FUNCTION_BLOCK ABSTRACT PiperModule IMPLEMENTS IPiperModule, ISequence, IStepManager
VAR
    _piperModule : PiperModuleInternal;
    i_sequence : SequenceType;
    _sequence : Sequencer(THIS^);
    command : PLCopenCall;
END_VAR

// Copyright (c) 2024 Loupe (https://loupe.team), provided under the MIT License.

METHOD _RequestStep : BOOL
VAR_INPUT
    nextStep : ENUM;
END_VAR
// Copyright (c) 2024 Loupe (https://loupe.team), provided under the MIT License.

_piperModule.requestSubstate := nextStep;
_piperModule.response := RESPONSE_STATE.BUSY;
_piperModule.requestNumber := _piperModule.requestNumber + 1;
END_METHOD

METHOD _Reset : BOOL
// Copyright (c) 2024 Loupe (https://loupe.team), provided under the MIT License.
END_METHOD

METHOD _SequenceComplete : BOOL
// Copyright (c) 2024 Loupe (https://loupe.team), provided under the MIT License.

_piperModule.requestSubstate := 0;
_piperModule.response := RESPONSE_STATE.DONE;
END_METHOD

METHOD _SequenceError : BOOL
// Copyright (c) 2024 Loupe (https://loupe.team), provided under the MIT License.

_piperModule.requestSubstate := 0;
_piperModule.response := RESPONSE_STATE.ERROR;
END_METHOD

METHOD Aborted : BOOL
// Copyright (c) 2024 Loupe (https://loupe.team), provided under the MIT License.

i_sequence.activeTasks.Aborted();
END_METHOD

METHOD Aborting : MACHINE_STATE
// Copyright (c) 2024 Loupe (https://loupe.team), provided under the MIT License.

_piperModule.skipsSync.aborting := TRUE;
END_METHOD

METHOD AbortingAsync : MACHINE_STATE
// Copyright (c) 2024 Loupe (https://loupe.team), provided under the MIT License.

_piperModule.skipsAsync.aborting := TRUE;
END_METHOD

METHOD Booting : MACHINE_STATE
// Copyright (c) 2024 Loupe (https://loupe.team), provided under the MIT License.

_piperModule.skipsSync.booting := TRUE;
END_METHOD

METHOD BootingAsync : MACHINE_STATE
// Copyright (c) 2024 Loupe (https://loupe.team), provided under the MIT License.

_piperModule.skipsAsync.booting := TRUE;
END_METHOD

METHOD CallState : BOOL
VAR_INPUT

END_VAR
// Copyright (c) 2024 Loupe (https://loupe.team), provided under the MIT License.

THIS^.WillCall();

IF THIS^._piperModule.previousSubstate <> THIS^.CurrentSubstate THEN
    THIS^.WillChangeSubstate();
END_IF

THIS^._piperModule.previousSubstate := THIS^.CurrentSubstate;

IF Response <> RESPONSE_STATE.DONE AND RequestedSubstate <= CurrentSubstate THEN
    CASE CurrentState OF
        MACHINE_STATE.ABORTING:
            IF NOT _piperModule.skipsSync.aborting THEN
                THIS^.Aborting();
            END_IF

        MACHINE_STATE.BOOTING:
            IF NOT _piperModule.skipsSync.booting THEN
                THIS^.Booting();
            END_IF

        MACHINE_STATE.CLEARING:
            IF NOT _piperModule.skipsSync.clearing THEN
                THIS^.Clearing();
            END_IF

        MACHINE_STATE.COMPLETING:
            IF NOT _piperModule.skipsSync.completing THEN
                THIS^.COMPLETING();
            END_IF

        MACHINE_STATE.EXECUTING:
            IF NOT _piperModule.skipsSync.executing THEN
                THIS^.Executing();
            END_IF

        MACHINE_STATE.HOLDING:
            IF NOT _piperModule.skipsSync.holding THEN
                THIS^.Holding();
            END_IF

        MACHINE_STATE.RESETTING:
            IF NOT _piperModule.skipsSync.resetting THEN
                THIS^.Resetting();
            END_IF

        MACHINE_STATE.STARTING:
            IF NOT _piperModule.skipsSync.starting THEN
                THIS^.Starting();
            END_IF

        MACHINE_STATE.STOPPING:
            IF NOT _piperModule.skipsSync.stopping THEN
                THIS^.Stopping();
            END_IF

        MACHINE_STATE.SUSPENDING:
            IF NOT _piperModule.skipsSync.suspending THEN
                THIS^.Suspending();
            END_IF

        MACHINE_STATE.UNHOLDING:
            IF NOT _piperModule.skipsSync.unholding THEN
                THIS^.Unholding();
            END_IF

        MACHINE_STATE.UNSUSPENDING:
            IF NOT _piperModule.skipsSync.unsuspending THEN
                THIS^.Unsuspending();
            END_IF

    END_CASE
END_IF

THIS^.DidCall();
END_METHOD

METHOD CallStateAsync : BOOL
VAR_INPUT

END_VAR
// Copyright (c) 2024 Loupe (https://loupe.team), provided under the MIT License.

THIS^.WillCallAsync();

IF THIS^._piperModule.previousSubstateAsync <> THIS^.CurrentSubstate THEN
    THIS^.WillChangeSubstateAsync();
END_IF

THIS^._piperModule.previousSubstateAsync := THIS^.CurrentSubstate;

IF Response <> RESPONSE_STATE.DONE AND RequestedSubstate <= CurrentSubstate THEN
    CASE CurrentState OF
        MACHINE_STATE.ABORTING:
            IF NOT _piperModule.skipsAsync.aborting THEN
                THIS^.AbortingAsync();
            ELSIF _piperModule.skipsSync.aborting THEN
                _piperModule.response := RESPONSE_STATE.DONE;
            END_IF

        MACHINE_STATE.BOOTING:
            IF NOT _piperModule.skipsAsync.booting THEN
                THIS^.BootingAsync();
            ELSIF _piperModule.skipsSync.booting THEN
                _piperModule.response := RESPONSE_STATE.DONE;
            END_IF

        MACHINE_STATE.CLEARING:
            IF NOT _piperModule.skipsAsync.clearing THEN
                THIS^.ClearingAsync();
            ELSIF _piperModule.skipsSync.clearing THEN
                _piperModule.response := RESPONSE_STATE.DONE;
            END_IF

        MACHINE_STATE.COMPLETING:
            IF NOT _piperModule.skipsAsync.completing THEN
                THIS^.CompletingAsync();
            ELSIF _piperModule.skipsSync.completing THEN
                _piperModule.response := RESPONSE_STATE.DONE;
            END_IF

        MACHINE_STATE.EXECUTING:
            IF NOT _piperModule.skipsAsync.executing THEN
                THIS^.ExecutingAsync();
            ELSIF _piperModule.skipsSync.executing THEN
                _piperModule.response := RESPONSE_STATE.DONE;
            END_IF

        MACHINE_STATE.HOLDING:
            IF NOT _piperModule.skipsAsync.holding THEN
                THIS^.HoldingAsync();
            ELSIF _piperModule.skipsSync.holding THEN
                _piperModule.response := RESPONSE_STATE.DONE;
            END_IF

        MACHINE_STATE.RESETTING:
            IF NOT _piperModule.skipsAsync.resetting THEN
                THIS^.ResettingAsync();
            ELSIF _piperModule.skipsSync.resetting THEN
                _piperModule.response := RESPONSE_STATE.DONE;
            END_IF

        MACHINE_STATE.STARTING:
            IF NOT _piperModule.skipsAsync.starting THEN
                THIS^.StartingAsync();
            ELSIF _piperModule.skipsSync.starting THEN
                _piperModule.response := RESPONSE_STATE.DONE;
            END_IF

        MACHINE_STATE.STOPPING:
            IF NOT _piperModule.skipsAsync.stopping THEN
                THIS^.StoppingAsync();
            ELSIF _piperModule.skipsSync.stopping THEN
                _piperModule.response := RESPONSE_STATE.DONE;
            END_IF

        MACHINE_STATE.SUSPENDING:
            IF NOT _piperModule.skipsAsync.suspending THEN
                THIS^.SuspendingAsync();
            ELSIF _piperModule.skipsSync.suspending THEN
                _piperModule.response := RESPONSE_STATE.DONE;
            END_IF

        MACHINE_STATE.UNHOLDING:
            IF NOT _piperModule.skipsAsync.unholding THEN
                THIS^.UnholdingAsync();
            ELSIF _piperModule.skipsSync.unholding THEN
                _piperModule.response := RESPONSE_STATE.DONE;
            END_IF

        MACHINE_STATE.UNSUSPENDING:
            IF NOT _piperModule.skipsAsync.unsuspending THEN
                THIS^.UnsuspendingAsync();
            ELSIF _piperModule.skipsSync.unsuspending THEN
                _piperModule.response := RESPONSE_STATE.DONE;
            END_IF

    END_CASE
END_IF

THIS^.DidCallAsync();
END_METHOD

METHOD PRIVATE CheckStatus : BOOL
VAR
    _commandIndex : INT;
    _anyAbort : BOOL;
    _anyBusy : BOOL;
    _anyError : BOOL;
END_VAR
// Copyright (c) 2024 Loupe (https://loupe.team), provided under the MIT License.

IF NOT i_sequence.statusChecked THEN
    //We cache the is abort so that we have a consistent 
    //	status for the whole state
    i_sequence.isError := i_sequence.activeTasks.isError;
    i_sequence.isAbort := i_sequence.activeTasks.isAbort;
    i_sequence.isDone := i_sequence.activeTasks.isDone;
END_IF
END_METHOD

METHOD Clearing : MACHINE_STATE
// Copyright (c) 2024 Loupe (https://loupe.team), provided under the MIT License.

_piperModule.skipsSync.clearing := TRUE;
END_METHOD

METHOD ClearingAsync : MACHINE_STATE
// Copyright (c) 2024 Loupe (https://loupe.team), provided under the MIT License.

_piperModule.skipsAsync.clearing := TRUE;
END_METHOD

METHOD Completing : MACHINE_STATE
// Copyright (c) 2024 Loupe (https://loupe.team), provided under the MIT License.

_piperModule.skipsSync.completing := TRUE;
END_METHOD

METHOD CompletingAsync : MACHINE_STATE
// Copyright (c) 2024 Loupe (https://loupe.team), provided under the MIT License.

_piperModule.skipsAsync.completing := TRUE;
END_METHOD

PROPERTY CurrentState : MACHINE_STATE
GET
// Copyright (c) 2024 Loupe (https://loupe.team), provided under the MIT License.

CurrentState := _piperModule.machine.PackMLState;
END_GET
END_PROPERTY

PROPERTY CurrentStep : ENUM
GET
// Copyright (c) 2024 Loupe (https://loupe.team), provided under the MIT License.

CurrentStep := ULINT_TO_UDINT(_piperModule.machine.Substate);
END_GET
END_PROPERTY

PROPERTY CurrentSubstate : ULINT
GET
// Copyright (c) 2024 Loupe (https://loupe.team), provided under the MIT License.

CurrentSubstate := _piperModule.machine.Substate;
END_GET
END_PROPERTY

METHOD DidCall : BOOL
VAR_INPUT
END_VAR
// Copyright (c) 2024 Loupe (https://loupe.team), provided under the MIT License.
END_METHOD

METHOD DidCallAsync : BOOL
VAR_INPUT
END_VAR
// Copyright (c) 2024 Loupe (https://loupe.team), provided under the MIT License.
END_METHOD

METHOD DoStep : ENUM
VAR
END_VAR
// Copyright (c) 2024 Loupe (https://loupe.team), provided under the MIT License.

DoStep := _sequence.DoStep();
END_METHOD

METHOD Errored : BOOL
VAR_INPUT
    ID : INT;
END_VAR
// Copyright (c) 2024 Loupe (https://loupe.team), provided under the MIT License.

i_sequence.activeTasks.Errored(ID);
END_METHOD

METHOD Executing : MACHINE_STATE
// Copyright (c) 2024 Loupe (https://loupe.team), provided under the MIT License.

_piperModule.skipsSync.executing := TRUE;
END_METHOD

METHOD ExecutingAsync : MACHINE_STATE
// Copyright (c) 2024 Loupe (https://loupe.team), provided under the MIT License.

_piperModule.skipsAsync.executing := TRUE;
END_METHOD

METHOD FB_init : BOOL
VAR_INPUT
    bInitRetains : BOOL; // if TRUE, the retain variables are initialized (warm start / cold start)
    bInCopyCode : BOOL; // if TRUE, the instance afterwards gets moved into the copy code (online change)
    machineIn : REFERENCE TO Piper;
    //	context : IPluginRunner;
END_VAR
// Copyright (c) 2024 Loupe (https://loupe.team), provided under the MIT License.
RegisterToMachine(machineIn);
//THIS^.setContext( context );
END_METHOD

METHOD Finished : BOOL
// Copyright (c) 2024 Loupe (https://loupe.team), provided under the MIT License.

i_sequence.activeTasks.Finished();
END_METHOD

METHOD Holding : MACHINE_STATE
// Copyright (c) 2024 Loupe (https://loupe.team), provided under the MIT License.

_piperModule.skipsSync.holding := TRUE;
END_METHOD

METHOD HoldingAsync : MACHINE_STATE
// Copyright (c) 2024 Loupe (https://loupe.team), provided under the MIT License.

_piperModule.skipsAsync.holding := TRUE;
END_METHOD

PROPERTY IsAbort : BOOL
GET
// Copyright (c) 2024 Loupe (https://loupe.team), provided under the MIT License.

CheckStatus();
IsAbort := i_sequence.isAbort;
END_GET
END_PROPERTY

PROPERTY IsDone : BOOL
GET
// Copyright (c) 2024 Loupe (https://loupe.team), provided under the MIT License.

CheckStatus();
IsDone := i_sequence.isDone;
END_GET
END_PROPERTY

PROPERTY IsError : BOOL
GET
// Copyright (c) 2024 Loupe (https://loupe.team), provided under the MIT License.

CheckStatus();
IsError := i_sequence.isError;
END_GET
END_PROPERTY

METHOD OnAbort : BOOL
VAR_INPUT
    nextStep : ENUM;
END_VAR
// Copyright (c) 2024 Loupe (https://loupe.team), provided under the MIT License.

OnAbort := _sequence.OnAbort(nextStep);
END_METHOD

METHOD OnEntry : BOOL
VAR_INPUT
END_VAR
// Copyright (c) 2024 Loupe (https://loupe.team), provided under the MIT License.

OnEntry := _sequence.OnEntry();
END_METHOD

METHOD OnError : BOOL
VAR_INPUT
    nextStep : ENUM;
END_VAR
// Copyright (c) 2024 Loupe (https://loupe.team), provided under the MIT License.

OnError := _sequence.OnError(nextStep);
END_METHOD

METHOD OnExit : BOOL
VAR_INPUT
END_VAR
// Copyright (c) 2024 Loupe (https://loupe.team), provided under the MIT License.

OnExit := _sequence.OnExit();
END_METHOD

METHOD OnFailure : BOOL
VAR_INPUT
    nextStep : ENUM;
END_VAR
// Copyright (c) 2024 Loupe (https://loupe.team), provided under the MIT License.

OnFailure := _sequence.OnFailure(nextStep);
END_METHOD

METHOD OnSuccess : BOOL
VAR_INPUT
    nextStep : ENUM;
END_VAR
// Copyright (c) 2024 Loupe (https://loupe.team), provided under the MIT License.

OnSuccess := _sequence.OnSuccess(nextStep);
END_METHOD

METHOD RegisterToMachine : DINT
VAR_INPUT
    machineIn : REFERENCE TO Piper;
END_VAR
VAR
END_VAR
// Copyright (c) 2024 Loupe (https://loupe.team), provided under the MIT License.
IF NOT _piperModule.registered THEN
    _piperModule.registered := TRUE;
    _piperModule.machine REF= machineIn;
    _piperModule.machine.RegisterSubmodule(THIS^);
END_IF
END_METHOD

{warning 'add property implementation'}
PROPERTY RequestedSubstate : ULINT
GET
// Copyright (c) 2024 Loupe (https://loupe.team), provided under the MIT License.

RequestedSubstate := _piperModule.requestSubstate;
END_GET
END_PROPERTY

PROPERTY RequestNumber : DINT
GET
// Copyright (c) 2024 Loupe (https://loupe.team), provided under the MIT License.

RequestNumber := _piperModule.requestNumber;
END_GET
END_PROPERTY

METHOD RequestStep : BOOL
VAR_INPUT
    nextStep : ENUM;
END_VAR
// Copyright (c) 2024 Loupe (https://loupe.team), provided under the MIT License.

RequestStep := _sequence.requestStep(nextStep);
END_METHOD

METHOD RequestStepClear : BOOL
VAR_INPUT
    nextStep : ENUM;
END_VAR
// Copyright (c) 2024 Loupe (https://loupe.team), provided under the MIT License.

RequestStepClear := _sequence.requestStepClear(nextStep);
END_METHOD

METHOD Resetting : BOOL
// Copyright (c) 2024 Loupe (https://loupe.team), provided under the MIT License.

_piperModule.skipsSync.resetting := TRUE;
END_METHOD

METHOD ResettingAsync : BOOL
// Copyright (c) 2024 Loupe (https://loupe.team), provided under the MIT License.

_piperModule.skipsAsync.resetting := TRUE;
END_METHOD

PROPERTY Response : RESPONSE_STATE
GET
// Copyright (c) 2024 Loupe (https://loupe.team), provided under the MIT License.

Response := _piperModule.response;
END_GET
END_PROPERTY

METHOD Run : BOOL
// Copyright (c) 2024 Loupe (https://loupe.team), provided under the MIT License.

THIS^.CallState();
END_METHOD

METHOD SequenceAbort : BOOL
VAR_INPUT
    ErrorCode : DINT;
    ErrorMessage : STRING;
END_VAR
// Copyright (c) 2024 Loupe (https://loupe.team), provided under the MIT License.

SequenceAbort := _sequence.sequenceAbort(ErrorCode, ErrorMessage);
END_METHOD

METHOD SequenceComplete : BOOL
VAR_INPUT
END_VAR
// Copyright (c) 2024 Loupe (https://loupe.team), provided under the MIT License.

SequenceComplete := _sequence.sequenceComplete();
END_METHOD

METHOD SequenceError : BOOL
VAR_INPUT
    ErrorCode : DINT;
    ErrorMessage : STRING;
END_VAR
// Copyright (c) 2024 Loupe (https://loupe.team), provided under the MIT License.

SequenceError := _sequence.sequenceError(ErrorCode, ErrorMessage);
END_METHOD

METHOD SetContext : BOOL
VAR_INPUT
    context : IPluginRunner;
END_VAR
// Copyright (c) 2024 Loupe (https://loupe.team), provided under the MIT License.
_piperModule.context := context;
context.RegisterPlugin(THIS^);
END_METHOD

METHOD SetState : BOOL
VAR_INPUT
END_VAR
// Copyright (c) 2024 Loupe (https://loupe.team), provided under the MIT License.

_piperModule.requestSubstate := 0;
_piperModule.response := RESPONSE_STATE.UNDEFINED;
_sequence.startSequence();
END_METHOD

METHOD Start : BOOL
VAR_INPUT
    Command : IPLCopenCommand;
END_VAR
// Copyright (c) 2024 Loupe (https://loupe.team), provided under the MIT License.

IF i_sequence.activeTasks.Start(Command) = 0 THEN
    //TODO: All out of commands.. Throw an error
    SequenceError(10000, 'Too Many Commands in 1 step');
    Start := FALSE;
ELSE
    Start := TRUE;
END_IF
END_METHOD

METHOD Starting : MACHINE_STATE
// Copyright (c) 2024 Loupe (https://loupe.team), provided under the MIT License.

_piperModule.skipsSync.starting := TRUE;
END_METHOD

METHOD StartingAsync : MACHINE_STATE
// Copyright (c) 2024 Loupe (https://loupe.team), provided under the MIT License.

_piperModule.skipsAsync.starting := TRUE;
END_METHOD

METHOD StartSequence : BOOL
// Copyright (c) 2024 Loupe (https://loupe.team), provided under the MIT License.

RequestStep(0);
END_METHOD

METHOD StateCompletePending : BOOL
VAR_INPUT
END_VAR
// Copyright (c) 2024 Loupe (https://loupe.team), provided under the MIT License.

_piperModule.response := RESPONSE_STATE.DONE_PENDING;
END_METHOD

METHOD StateErrored : BOOL
VAR_INPUT
END_VAR
// Copyright (c) 2024 Loupe (https://loupe.team), provided under the MIT License.

_piperModule.response := RESPONSE_STATE.ERROR;
END_METHOD

METHOD Stopping : MACHINE_STATE
// Copyright (c) 2024 Loupe (https://loupe.team), provided under the MIT License.

_piperModule.skipsSync.stopping := TRUE;
END_METHOD

METHOD StoppingAsync : MACHINE_STATE
// Copyright (c) 2024 Loupe (https://loupe.team), provided under the MIT License.

_piperModule.skipsAsync.stopping := TRUE;
END_METHOD

METHOD Suspending : MACHINE_STATE
// Copyright (c) 2024 Loupe (https://loupe.team), provided under the MIT License.

_piperModule.skipsSync.suspending := TRUE;
END_METHOD

METHOD SuspendingAsync : MACHINE_STATE
// Copyright (c) 2024 Loupe (https://loupe.team), provided under the MIT License.

_piperModule.skipsAsync.suspending := TRUE;
END_METHOD

METHOD Undefined : MACHINE_STATE
// Copyright (c) 2024 Loupe (https://loupe.team), provided under the MIT License.

_piperModule.response := RESPONSE_STATE.NO_IMPL;
END_METHOD

METHOD UndefinedAsync : MACHINE_STATE
// Copyright (c) 2024 Loupe (https://loupe.team), provided under the MIT License.
END_METHOD

METHOD Unholding : MACHINE_STATE
// Copyright (c) 2024 Loupe (https://loupe.team), provided under the MIT License.

_piperModule.skipsSync.unholding := TRUE;
END_METHOD

METHOD UnholdingAsync : MACHINE_STATE
// Copyright (c) 2024 Loupe (https://loupe.team), provided under the MIT License.

_piperModule.skipsAsync.unholding := TRUE;
END_METHOD

METHOD Unsuspending : MACHINE_STATE
// Copyright (c) 2024 Loupe (https://loupe.team), provided under the MIT License.

_piperModule.skipsSync.unsuspending := TRUE;
END_METHOD

METHOD UnsuspendingAsync : MACHINE_STATE
// Copyright (c) 2024 Loupe (https://loupe.team), provided under the MIT License.

_piperModule.skipsAsync.unsuspending := TRUE;
END_METHOD

METHOD WillCall : BOOL
VAR_INPUT
END_VAR
// Copyright (c) 2024 Loupe (https://loupe.team), provided under the MIT License.
END_METHOD

METHOD WillCallAsync : BOOL
VAR_INPUT
END_VAR
// Copyright (c) 2024 Loupe (https://loupe.team), provided under the MIT License.
END_METHOD

METHOD WillChangeSubstate : BOOL
VAR_INPUT
END_VAR
// Copyright (c) 2024 Loupe (https://loupe.team), provided under the MIT License.
END_METHOD

METHOD WillChangeSubstateAsync : BOOL
VAR_INPUT
END_VAR
// Copyright (c) 2024 Loupe (https://loupe.team), provided under the MIT License.
END_METHOD

END_FUNCTION_BLOCK

(* stored: Version 1.1.0.1
   POU PiperModule: Id {a49f2d62-e1fb-48a5-85f3-63c6ca0008b5}, SpecialFunc None
   Folder Handshake: Id {4c5f2be6-50e2-4221-9823-927772de0d3d}
   Folder PackML: Id {103dd83a-b3d9-4ad0-8c08-4f9980ee4239}
   Folder PackMLAsync: Id {8d7f90b0-8dd2-435c-bd8c-5cc1b1fbb6fd}
   Folder PLCopen: Id {64089310-c2b2-409b-a0ee-99363ab988ef}
   Folder Sequence: Id {8453be56-3070-4e48-be57-e6bddaa0c622}
   Folder callbacks: Id {778d4fd5-4d6a-48ab-b39c-efcbe9f36276}
   Folder StateControl: Id {6b001fba-3153-4b1f-932c-0a719f676126}
   Folder Setup: Id {eeb68776-0e62-46f1-9ad5-da0f6ad004d6}
   Folder StepManager: Id {48dc10ce-7eca-4656-a440-fb808be36402}
   Method _RequestStep: Id {f4f6af93-0cb3-42b4-9ca9-21e1cca56843}
   Method _Reset: Id {e5c4fbde-1df8-48bc-9d3c-c9ad0b85ba57}
   Method _SequenceComplete: Id {93d7990e-83cd-41da-874b-7bcab730bc0b}
   Method _SequenceError: Id {d8c3afc4-de9e-411e-b9c4-728f5280910b}
   Method Aborted: Id {bfc1fdac-439e-4113-ad1e-f9923d22408a}
   Method Aborting: Id {f8a973b9-f9f6-410e-b5c1-d3a51e04d7ba}
   Method AbortingAsync: Id {cec06300-8aeb-4e42-9276-4c70e9317f91}
   Method Booting: Id {8c4cd35b-8b79-4b7d-b8d1-be00bdf7a998}
   Method BootingAsync: Id {9ce4a9c1-65bb-4257-8807-dd0b22b34a12}
   Method CallState: Id {8c189048-9fa3-4697-bf51-2b2792a9dbd0}
   Method CallStateAsync: Id {e1b90424-eb8a-4298-af7b-9ebf7a18fd7f}
   Method CheckStatus: Id {86f2cd85-d973-4227-9da3-ee4c3ed52cb2}
   Method Clearing: Id {7bee31c9-141c-4358-8aca-33cad167ec8c}
   Method ClearingAsync: Id {f3e36a82-f507-456f-b94b-64cf7681213f}
   Method Completing: Id {a413a61c-6ca7-4fd3-9296-7d7fa43065a1}
   Method CompletingAsync: Id {a25aad53-5324-4bcd-8931-defa299aa789}
   Property CurrentState: Id {a9acd7a7-2c0b-4c94-b2f1-fd8eff4ca549}
   Get Get: Id {f9b34f5c-82e0-4f78-84c5-ae373d09c208}
   Property CurrentStep: Id {674ced14-3f04-4cfd-8fdd-09d4136719f6}
   Get Get: Id {bf1b5077-fd19-49ed-99c4-4f1808c79d8e}
   Property CurrentSubstate: Id {88b27a69-ed23-442a-a3ec-53bdad984f5d}
   Get Get: Id {b3583fbe-c993-43b1-b2df-a70ec57198b2}
   Method DidCall: Id {5d73cdfc-bb8e-4ce5-9441-fb7bff95dddb}
   Method DidCallAsync: Id {1c612e8f-0b57-4feb-b3a0-8272535d9fbf}
   Method DoStep: Id {2460656a-9a34-4d02-b4bf-86513714621e}
   Method Errored: Id {06792213-1d5a-46af-b439-4e2d3ae32a97}
   Method Executing: Id {7d2b0e0c-1f31-466b-8d1a-373403d052a1}
   Method ExecutingAsync: Id {f195c071-1809-4503-9600-76c76102562b}
   Method FB_Init: Id {44756489-9d5d-4428-aeab-3bb684fa1b7a}
   Method Finished: Id {c79313eb-7bb8-4f2e-95d1-b7033d0c3362}
   Method Holding: Id {894a69b8-8e15-4bf4-acd5-ce7c5d137725}
   Method HoldingAsync: Id {c029deb6-41db-4d4c-af7b-1fd6e8644624}
   Property IsAbort: Id {2dcca336-a4f0-4f55-9876-b7ff3b24f026}
   Get Get: Id {e020552a-3b08-4a7b-876e-0e16adbd262f}
   Property IsDone: Id {af18764f-0737-410b-95a0-2ab146c203c3}
   Get Get: Id {86cfcbf8-6913-4a08-a2cd-03f06f59d324}
   Property IsError: Id {ccf11f90-16bd-4026-9f26-622caad6e51f}
   Get Get: Id {ac9dcd1c-2e71-4438-99fd-7782403a6099}
   Method OnAbort: Id {516af93a-5d99-4bdf-960c-3294b3cb47e0}
   Method OnEntry: Id {6689b526-5baa-4f23-b571-4ec7663af97d}
   Method OnError: Id {3514fd98-aade-49a4-8005-f8ef205958d8}
   Method OnExit: Id {73e201fe-6ff5-45dc-ba48-16917ae7f7e3}
   Method OnFailure: Id {3f9573b7-b22b-45b2-a5b3-ac03573adb91}
   Method OnSuccess: Id {2218590e-0706-443f-94cd-47156df6e0ea}
   Method RegisterToMachine: Id {3f378610-e9ba-4ac4-ba6e-e297be53cd18}
   Property RequestedSubstate: Id {ca192a6a-e2d8-4eec-8bb5-126fe0cbacbb}
   Get Get: Id {b76addb0-caf3-43be-a1d2-774e6ae0391a}
   Property RequestNumber: Id {603863d1-8473-47c0-b2ce-fa34eb6e2919}
   Get Get: Id {d46e1119-18d1-4a0c-ad96-ef1cba488e1d}
   Method RequestStep: Id {0e4176a8-3797-4a27-9ba5-06223fd5ae03}
   Method RequestStepClear: Id {e97e13d9-69d6-493d-a91f-a645bb23f6bb}
   Method Resetting: Id {d15239fc-c709-4b5f-b06c-c65056e3acbe}
   Method ResettingAsync: Id {f993b6c7-b4af-4377-a0d6-8a2380615fa3}
   Property Response: Id {8eb07caf-319e-4b96-aa33-5592ef7d8262}
   Get Get: Id {403fda28-4e41-44b0-8df2-3a36eb884c0a}
   Method Run: Id {403e4da3-736c-4b46-bfe8-d21525e61697}
   Method SequenceAbort: Id {382ae541-7c29-4690-b84d-2cbc2d1546e3}
   Method SequenceComplete: Id {e7a11495-e96e-44f3-b8dd-fb20c40130d2}
   Method SequenceError: Id {6e2cc27d-5672-4397-b236-2cd116232adf}
   Method SetContext: Id {f6595b8f-ae99-4b2e-85fc-1c2a518ea4e4}
   Method SetState: Id {86fb48a2-6e78-48ff-9d41-f8e50cfe20ac}
   Method Start: Id {0fbe109f-325f-4002-b69e-be08f70d2754}
   Method Starting: Id {a86c3956-3fb4-4d94-b103-59d08284b030}
   Method StartingAsync: Id {f0a9676d-2362-4f42-9b4a-07835a470b0e}
   Method StartSequence: Id {cf35b5b2-fbce-4fdb-a962-ec55492f889b}
   Method StateCompletePending: Id {3c3f8f98-6626-4764-a216-4b263314b59d}
   Method StateErrored: Id {3ac147a4-b6ee-453f-bca1-363fc1d7eaed}
   Method Stopping: Id {301f156c-360f-470c-88cd-689b56d4fe1f}
   Method StoppingAsync: Id {ecb23d71-1a43-461c-aa40-2add24e1194d}
   Method Suspending: Id {bf1c4eed-ae50-4104-8c79-3a268c628404}
   Method SuspendingAsync: Id {f3583032-054c-4d43-8d68-39f2c7f4866f}
   Method Undefined: Id {dce2f0f3-de0c-4095-9eb2-087dc401d55d}
   Method UndefinedAsync: Id {df63348c-7f98-4cdb-8860-51cf22a0da80}
   Method Unholding: Id {3eb5a5dc-5d0d-486e-947a-67764a0c3038}
   Method UnholdingAsync: Id {d6a9e8cc-d336-42ad-8812-a767d9f87070}
   Method Unsuspending: Id {d7a887dc-24e3-45a9-bfab-9b8c964676e6}
   Method UnsuspendingAsync: Id {b8341822-21e7-482e-b82c-93c76e5c31dc}
   Method WillCall: Id {e88ecae5-093b-4df2-8a31-55fa62529e6c}
   Method WillCallAsync: Id {3da853bb-6490-4d04-a4d1-57912c1a0048}
   Method WillChangeSubstate: Id {7dcc840a-b340-4d0d-8cb4-fe075b5c4c05}
   Method WillChangeSubstateAsync: Id {538c49c4-4889-4a9f-b501-4dace4dcbf3f} *)
